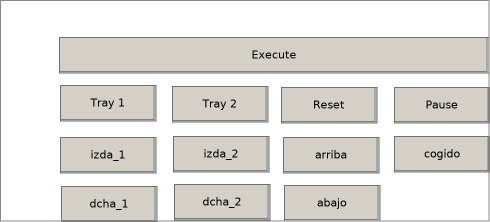
VISUALIZATION Visualization  // 490x222
    Button (59,37 430x36), "Execute"
        tap MAIN.Controller.Execute
    Button (60,85 96x36), "Tray 1"
        tap MAIN.Controller.Tray_1
    Button (172,86 96x36), "Tray 2"
        tap MAIN.Controller.Tray_2
    Button (60,137 96x36), "izda_1"
        toggle MAIN.Controller.Discharger.izda_1
    Button (173,136 96x36), "izda_2"
        toggle MAIN.Controller.Discharger.izda_2
    Button (283,137 96x36), "arriba"
        toggle MAIN.Controller.Discharger.arriba
    Button (394,136 96x36), "cogido"
        toggle MAIN.Controller.Discharger.cogido
    Button (281,87 96x36), "Reset"
        tap MAIN.Controller.Reset
    Button (394,87 96x36), "Pause"
        tap MAIN.Controller.Pause
    Button (61,186 96x36), "dcha_1"
        toggle MAIN.Controller.Discharger.dcha_1
    Button (174,184 96x36), "dcha_2"
        toggle MAIN.Controller.Discharger.dcha_2
    Button (284,185 96x36), "abajo"
        toggle MAIN.Controller.Discharger.abajo
END_VISUALIZATION

(* stored: Version 1.1.0.1, ProductVersion 3.1.4024.6
   Visu Visualization: Id {ae0ba0af-939e-4a05-84b7-c64d8697f730} *)
